Fanuc KAREL source: KO00081.KL

PROGRAM KO00081
%NOLOCKGROUP
%ENVIRONMENT MIR
VAR
  P1: JOINTPOS
  P2: POSITION
  F: BOOLEAN
  OUT: POSITION
BEGIN
  F = TRUE
  OUT = MIRROR(P1, P2, F)
END KO00081
